Omron CX-Programmer project NewProject (CX-Programmer 9.73)

# PLC system: CP1L M

## Global symbols (name address type ; comment)
ALL_TANKS_ARE_FULL 102.04 BOOL  ; Cac thung day
AUTO 0.03 BOOL  ; Tu dong
C0004 BOOL  ; 1
D0 CHANNEL  ; COMPARE
D2 CHANNEL  ; .
BLOWER 100.00 BOOL  ; Lam sach
CHECK_1 1.10 BOOL  ; Kiem tra 1
CHECK_2 1.11 BOOL  ; Kiem tra 2
CHECK_3 2.00 BOOL  ; Kiem tra 3
CONVETOR_W2 101.02 BOOL  ; Chuyen doi 2
CONVEYOR_1 103.01 BOOL  ; Bang chuyen 1
CONVEYOR_10 103.09 BOOL  ; Bang chuyen 10
CONVEYOR_11 103.10 BOOL  ; Bang chuyen 11
CONVEYOR_2 103.02 BOOL  ; Bang chuyen 2
CONVEYOR_3 103.03 BOOL  ; Bang chuyen 3
CONVEYOR_5 103.04 BOOL  ; Bang chuyen 5
CONVEYOR_6 103.05 BOOL  ; Bang chuyen 6
CONVEYOR_7 103.06 BOOL  ; Bang chuyen 7
CONVEYOR_9 103.08 BOOL  ; Bang chuyen 9
CONVEYOR_W1 101.01 BOOL  ; Chuyen doi 1
CONVEYOR_W3 101.03 BOOL  ; Chuyen doi 3
DEFAULT_TANK_VOLUME 2.02 BOOL  ; Muc be mac dinh
DROP_1 101.04 BOOL  ; Tha 1
DROP_2 101.05 BOOL  ; Tha 2
DROP_3 101.06 BOOL  ; Tha 3
EJECT_BLOWER 100.01 BOOL  ; Ngung lam sach
EJECT_PRINT 100.04 BOOL  ; Ngung in
ERROR_LIGHT 101.00 BOOL  ; Den bao dong
KEEP_SENSOR_C1 102.03 BOOL  ; Giu cam bien 1
KEEP_SENSOR_C2 102.02 BOOL  ; Giu cam bien 2
KEEP_SENSOR_C3 102.01 BOOL  ; Giu cam bien 3
MANUAL 0.02 BOOL  ; In don chiec
METAL 2.06 BOOL  ; Kim loai
PAPER 2.07 BOOL  ; Giay
PLASTIC 2.08 BOOL  ; Nhua
POWER 103.00 BOOL  ; Nguon
PRINT_LIGHT 100.02 BOOL  ; In sang
PRINT_MACHINE 100.03 BOOL  ; In may
QUALITIFY_SENSOR 1.09 BOOL  ; Cam bien chat luong
REJECT 101.07 BOOL  ; Loai bo
REJECTED_PRODUCT 2.01 BOOL  ; San pham loi
REJECT_CONVEYOR 103.07 BOOL  ; Bang chuyen san pham loi
RESET_ALL 102.08 BOOL  ; Doi het cac thung
RESET_PACK_1 102.05 BOOL  ; Doi thung 1
RESET_PACK_2 102.06 BOOL  ; Doi thung 2
RESET_PACK_3 102.07 BOOL  ; Doi thung 3
ROBOT_CLA 102.00 BOOL  ; Canh tay robot
SENSOR_1 1.00 BOOL  ; Cam bien 1
SENSOR_2 1.01 BOOL  ; Cam bien 2
SENSOR_3 1.02 BOOL  ; Cam bien 3
SENSOR_4 1.03 BOOL  ; Cam bien 4
SENSOR_5 1.04 BOOL  ; Cam bien 5
SENSOR_6 1.05 BOOL  ; Cam bien 6
SENSOR_CLASSTIFY_1 1.08 BOOL  ; Cam bien phan loai 1
SENSOR_CLASSTIFY_2 1.07 BOOL  ; Cam bien phan loai 2
SENSOR_CLASSTIFY_3 1.06 BOOL  ; Cam bien phan loai 3
SENSOR_PACK_1 2.03 BOOL  ; Cam bien hang 1
SENSOR_PACK_2 2.04 BOOL  ; Cam bien hang 2
SENSOR_PACK_3 2.05 BOOL  ; Cam bien hang 3
START 0.00 BOOL  ; Nut khoi dong
STOP 0.01 BOOL  ; Nut dung
WAY_1 100.05 BOOL  ; Duong 1
WAY_2 100.06 BOOL  ; Duong 2
WAY_3 100.07 BOOL  ; Duong 3

## Program NewProgram1 (cyclic task 0)
Local symbols
dD0 UINT

### Section Section1

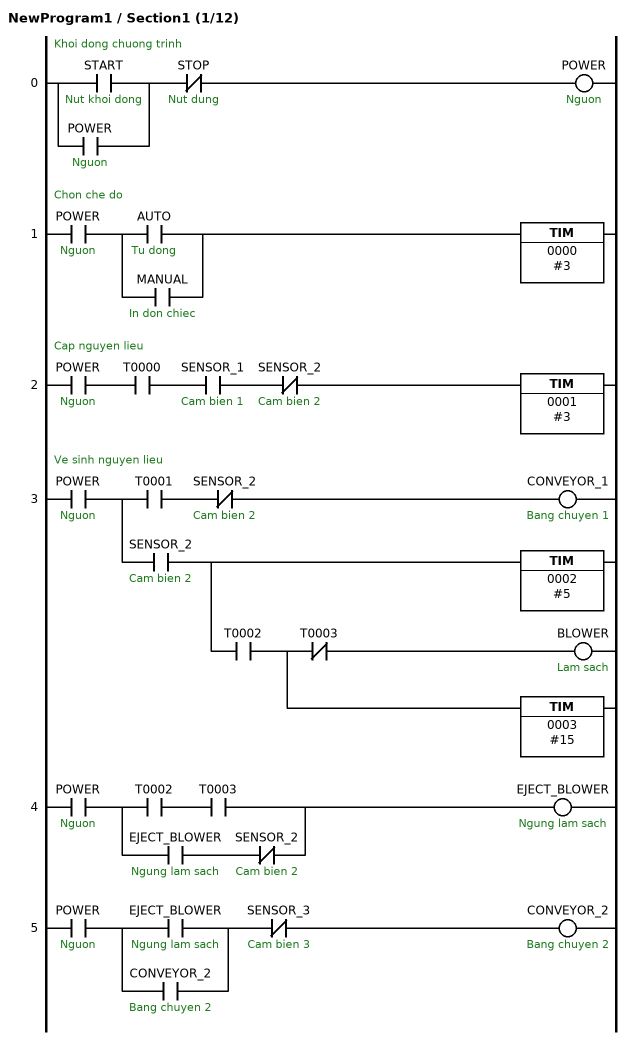
; rung 0: Khoi dong chuong trinh
LD START  ; Nut khoi dong
OR POWER  ; Nguon
ANDNOT STOP  ; Nut dung
OUT POWER  ; Nguon
; rung 1: Chon che do
LD POWER  ; Nguon
LD AUTO  ; Tu dong
OR MANUAL  ; In don chiec
ANDLD
TIM 0000 #3
; rung 2: Cap nguyen lieu
LD POWER  ; Nguon
AND T0000
AND SENSOR_1  ; Cam bien 1
ANDNOT SENSOR_2  ; Cam bien 2
TIM 0001 #3
; rung 3: Ve sinh nguyen lieu
LD POWER  ; Nguon
OUT TR0
AND T0001
ANDNOT SENSOR_2  ; Cam bien 2
OUT CONVEYOR_1  ; Bang chuyen 1
LD TR0
AND SENSOR_2  ; Cam bien 2
TIM 0002 #5
AND T0002
OUT TR0
ANDNOT T0003
OUT BLOWER  ; Lam sach
LD TR0
TIM 0003 #15
; rung 4
LD POWER  ; Nguon
LD T0002
AND T0003
LD EJECT_BLOWER  ; Ngung lam sach
ANDNOT SENSOR_2  ; Cam bien 2
ORLD
ANDLD
OUT EJECT_BLOWER  ; Ngung lam sach
; rung 5
LD POWER  ; Nguon
LD EJECT_BLOWER  ; Ngung lam sach
OR CONVEYOR_2  ; Bang chuyen 2
ANDLD
ANDNOT SENSOR_3  ; Cam bien 3
OUT CONVEYOR_2  ; Bang chuyen 2

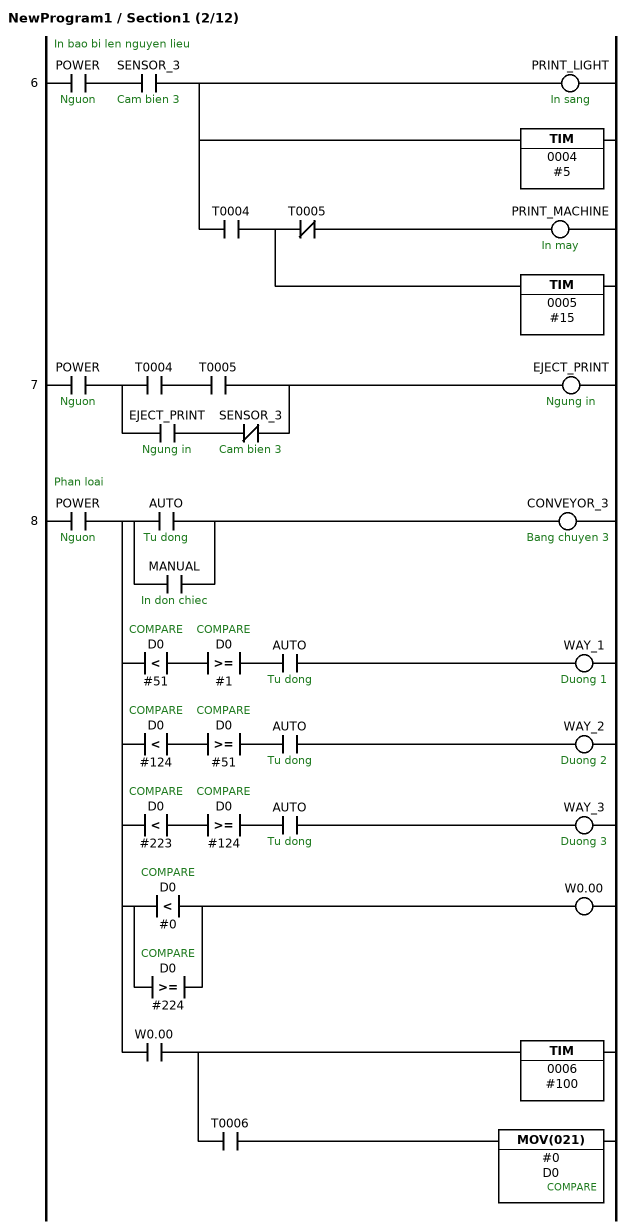
; rung 6: In bao bi len nguyen lieu
LD POWER  ; Nguon
AND SENSOR_3  ; Cam bien 3
OUT PRINT_LIGHT  ; In sang
TIM 0004 #5
AND T0004
OUT TR0
ANDNOT T0005
OUT PRINT_MACHINE  ; In may
LD TR0
TIM 0005 #15
; rung 7
LD POWER  ; Nguon
LD T0004
AND T0005
LD EJECT_PRINT  ; Ngung in
ANDNOT SENSOR_3  ; Cam bien 3
ORLD
ANDLD
OUT EJECT_PRINT  ; Ngung in
; rung 8: Phan loai
LD POWER  ; Nguon
OUT TR0
LD AUTO  ; Tu dong
OR MANUAL  ; In don chiec
ANDLD
OUT CONVEYOR_3  ; Bang chuyen 3
LD TR0
AND<(310) D0 #51  ; COMPARE
AND>=(325) D0 #1  ; COMPARE
AND AUTO  ; Tu dong
OUT WAY_1  ; Duong 1
LD TR0
AND<(310) D0 #124  ; COMPARE
AND>=(325) D0 #51  ; COMPARE
AND AUTO  ; Tu dong
OUT WAY_2  ; Duong 2
LD TR0
AND<(310) D0 #223  ; COMPARE
AND>=(325) D0 #124  ; COMPARE
AND AUTO  ; Tu dong
OUT WAY_3  ; Duong 3
LD TR0
LD<(310) D0 #0  ; COMPARE
OR>=(325) D0 #224  ; COMPARE
ANDLD
OUT W0.00
LD TR0
AND W0.00
TIM 0006 #100
AND T0006
MOV(021) #0 D0  ; COMPARE

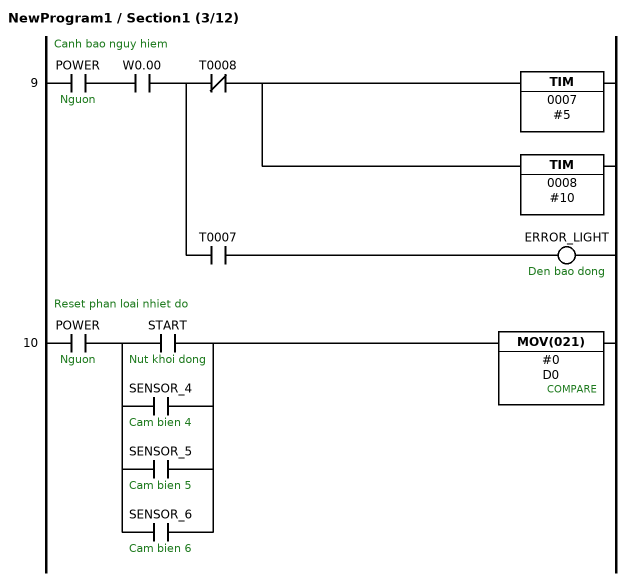
; rung 9: Canh bao nguy hiem
LD POWER  ; Nguon
AND W0.00
OUT TR0
ANDNOT T0008
TIM 0007 #5
TIM 0008 #10
LD TR0
AND T0007
OUT ERROR_LIGHT  ; Den bao dong
; rung 10: Reset phan loai nhiet do
LD POWER  ; Nguon
LD START  ; Nut khoi dong
OR SENSOR_4  ; Cam bien 4
OR SENSOR_5  ; Cam bien 5
OR SENSOR_6  ; Cam bien 6
ANDLD
MOV(021) #0 D0  ; COMPARE

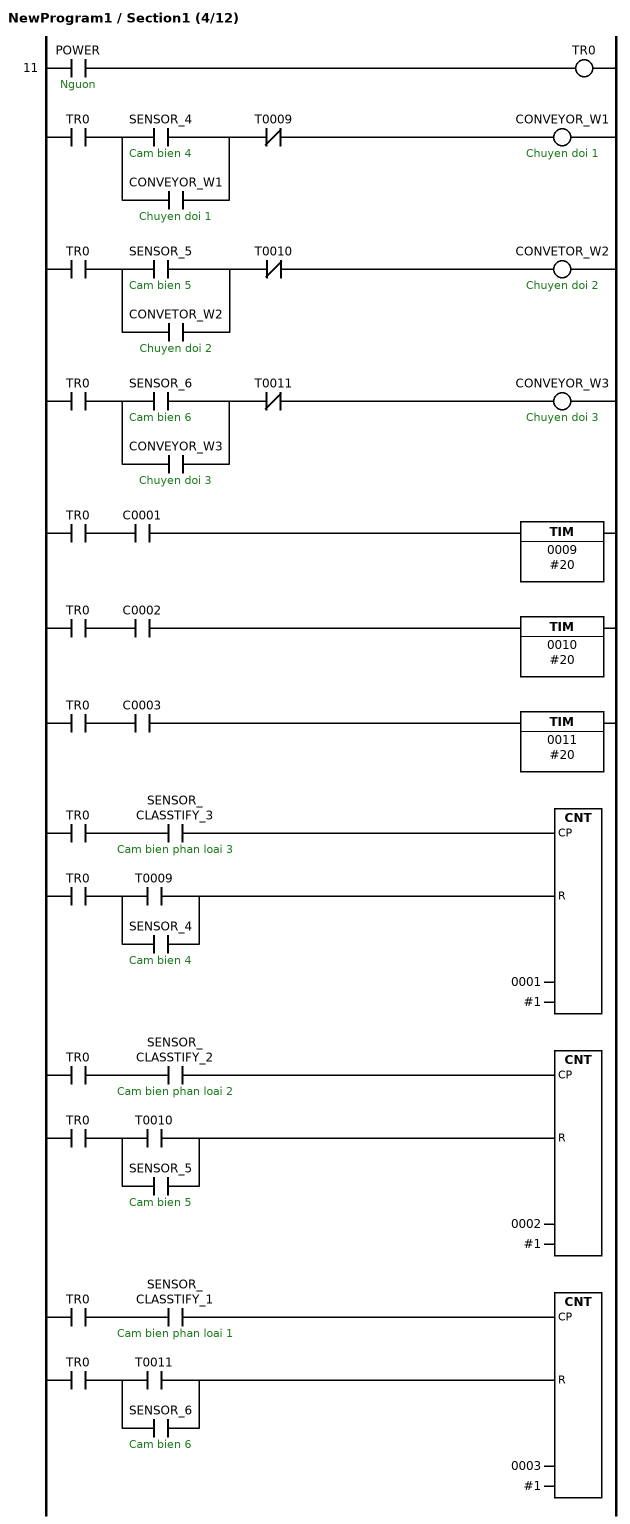
; rung 11
LD POWER  ; Nguon
OUT TR0
LD SENSOR_4  ; Cam bien 4
OR CONVEYOR_W1  ; Chuyen doi 1
ANDLD
ANDNOT T0009
OUT CONVEYOR_W1  ; Chuyen doi 1
LD TR0
LD SENSOR_5  ; Cam bien 5
OR CONVETOR_W2  ; Chuyen doi 2
ANDLD
ANDNOT T0010
OUT CONVETOR_W2  ; Chuyen doi 2
LD TR0
LD SENSOR_6  ; Cam bien 6
OR CONVEYOR_W3  ; Chuyen doi 3
ANDLD
ANDNOT T0011
OUT CONVEYOR_W3  ; Chuyen doi 3
LD TR0
AND C0001
TIM 0009 #20
LD TR0
AND C0002
TIM 0010 #20
LD TR0
AND C0003
TIM 0011 #20
LD TR0
AND SENSOR_CLASSTIFY_3  ; Cam bien phan loai 3
LD TR0
LD T0009
OR SENSOR_4  ; Cam bien 4
ANDLD
CNT 0001 #1
LD TR0
AND SENSOR_CLASSTIFY_2  ; Cam bien phan loai 2
LD TR0
LD T0010
OR SENSOR_5  ; Cam bien 5
ANDLD
CNT 0002 #1
LD TR0
AND SENSOR_CLASSTIFY_1  ; Cam bien phan loai 1
LD TR0
LD T0011
OR SENSOR_6  ; Cam bien 6
ANDLD
CNT 0003 #1

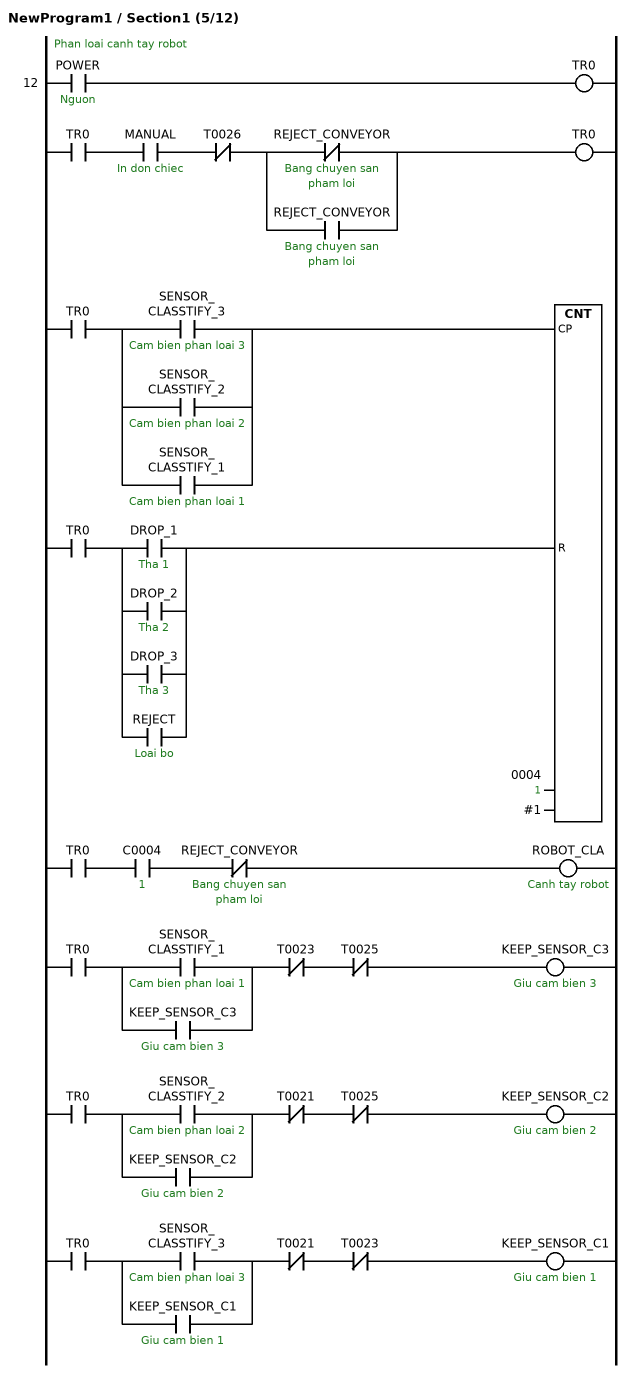
; rung 12: Phan loai canh tay robot
LD POWER  ; Nguon
OUT TR0
LD SENSOR_CLASSTIFY_3  ; Cam bien phan loai 3
OR SENSOR_CLASSTIFY_2  ; Cam bien phan loai 2
OR SENSOR_CLASSTIFY_1  ; Cam bien phan loai 1
ANDLD
LD TR0
LD DROP_1  ; Tha 1
OR DROP_2  ; Tha 2
OR DROP_3  ; Tha 3
OR REJECT  ; Loai bo
ANDLD
CNT 0004 #1  ; 1
LD TR0
AND C0004  ; 1
ANDNOT REJECT_CONVEYOR  ; Bang chuyen san pham loi
OUT ROBOT_CLA  ; Canh tay robot
LD TR0
AND MANUAL  ; In don chiec
ANDNOT T0026
LDNOT REJECT_CONVEYOR  ; Bang chuyen san pham loi
OR REJECT_CONVEYOR  ; Bang chuyen san pham loi
ANDLD
OUT TR0
LD SENSOR_CLASSTIFY_1  ; Cam bien phan loai 1
OR KEEP_SENSOR_C3  ; Giu cam bien 3
ANDLD
ANDNOT T0023
ANDNOT T0025
OUT KEEP_SENSOR_C3  ; Giu cam bien 3
LD TR0
LD SENSOR_CLASSTIFY_2  ; Cam bien phan loai 2
OR KEEP_SENSOR_C2  ; Giu cam bien 2
ANDLD
ANDNOT T0021
ANDNOT T0025
OUT KEEP_SENSOR_C2  ; Giu cam bien 2
LD TR0
LD SENSOR_CLASSTIFY_3  ; Cam bien phan loai 3
OR KEEP_SENSOR_C1  ; Giu cam bien 1
ANDLD
ANDNOT T0021
ANDNOT T0023
OUT KEEP_SENSOR_C1  ; Giu cam bien 1

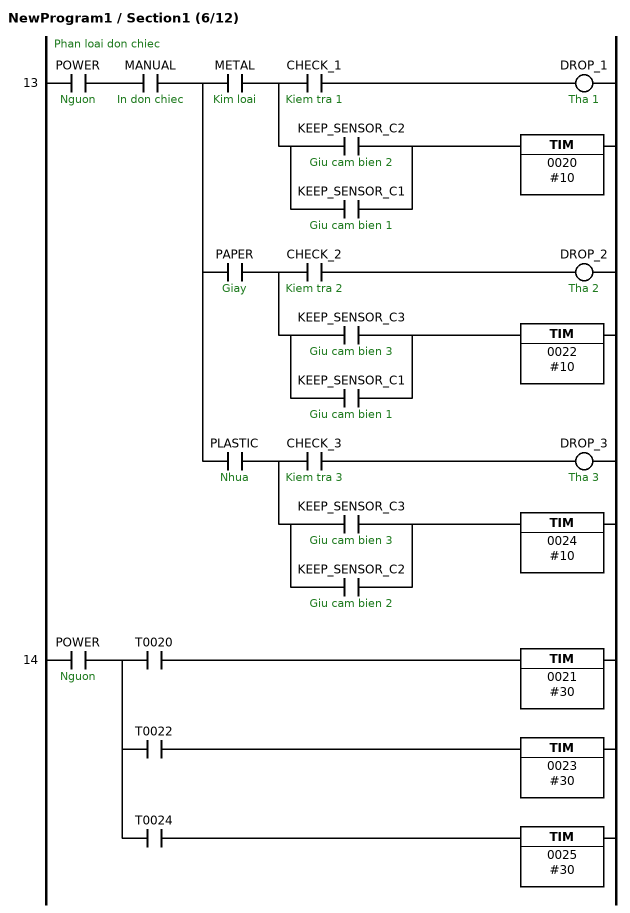
; rung 13: Phan loai don chiec
LD POWER  ; Nguon
AND MANUAL  ; In don chiec
OUT TR0
AND METAL  ; Kim loai
OUT TR1
AND CHECK_1  ; Kiem tra 1
OUT DROP_1  ; Tha 1
LD TR1
LD KEEP_SENSOR_C2  ; Giu cam bien 2
OR KEEP_SENSOR_C1  ; Giu cam bien 1
ANDLD
TIM 0020 #10
LD TR0
AND PAPER  ; Giay
OUT TR1
AND CHECK_2  ; Kiem tra 2
OUT DROP_2  ; Tha 2
LD TR1
LD KEEP_SENSOR_C3  ; Giu cam bien 3
OR KEEP_SENSOR_C1  ; Giu cam bien 1
ANDLD
TIM 0022 #10
LD TR0
AND PLASTIC  ; Nhua
OUT TR0
AND CHECK_3  ; Kiem tra 3
OUT DROP_3  ; Tha 3
LD TR0
LD KEEP_SENSOR_C3  ; Giu cam bien 3
OR KEEP_SENSOR_C2  ; Giu cam bien 2
ANDLD
TIM 0024 #10
; rung 14
LD POWER  ; Nguon
OUT TR0
AND T0020
TIM 0021 #30
LD TR0
AND T0022
TIM 0023 #30
LD TR0
AND T0024
TIM 0025 #30

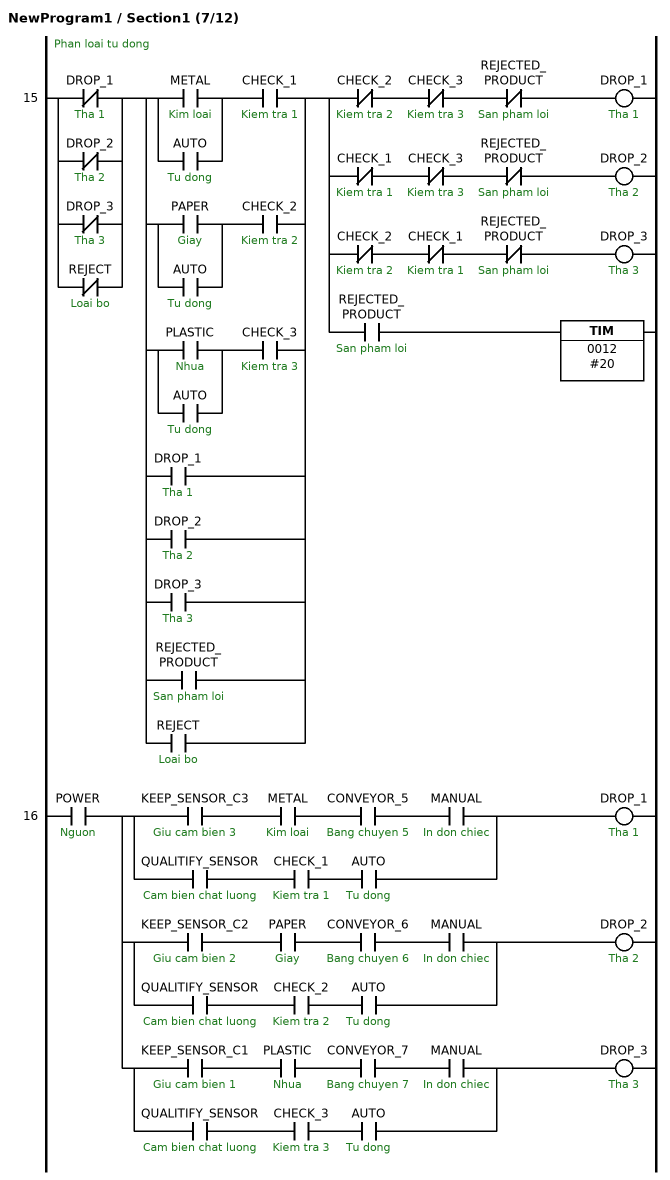
; rung 15: Phan loai tu dong
LDNOT DROP_1  ; Tha 1
ORNOT DROP_2  ; Tha 2
ORNOT DROP_3  ; Tha 3
ORNOT REJECT  ; Loai bo
LD METAL  ; Kim loai
OR AUTO  ; Tu dong
AND CHECK_1  ; Kiem tra 1
LD PAPER  ; Giay
OR AUTO  ; Tu dong
AND CHECK_2  ; Kiem tra 2
ORLD
LD PLASTIC  ; Nhua
OR AUTO  ; Tu dong
AND CHECK_3  ; Kiem tra 3
ORLD
OR DROP_1  ; Tha 1
OR DROP_2  ; Tha 2
OR DROP_3  ; Tha 3
OR REJECTED_PRODUCT  ; San pham loi
OR REJECT  ; Loai bo
ANDLD
OUT TR0
ANDNOT CHECK_2  ; Kiem tra 2
ANDNOT CHECK_3  ; Kiem tra 3
ANDNOT REJECTED_PRODUCT  ; San pham loi
OUT DROP_1  ; Tha 1
LD TR0
ANDNOT CHECK_1  ; Kiem tra 1
ANDNOT CHECK_3  ; Kiem tra 3
ANDNOT REJECTED_PRODUCT  ; San pham loi
OUT DROP_2  ; Tha 2
LD TR0
ANDNOT CHECK_2  ; Kiem tra 2
ANDNOT CHECK_1  ; Kiem tra 1
ANDNOT REJECTED_PRODUCT  ; San pham loi
OUT DROP_3  ; Tha 3
LD TR0
AND REJECTED_PRODUCT  ; San pham loi
TIM 0012 #20
; rung 16
LD POWER  ; Nguon
OUT TR0
LD KEEP_SENSOR_C3  ; Giu cam bien 3
AND METAL  ; Kim loai
AND CONVEYOR_5  ; Bang chuyen 5
AND MANUAL  ; In don chiec
LD QUALITIFY_SENSOR  ; Cam bien chat luong
AND CHECK_1  ; Kiem tra 1
AND AUTO  ; Tu dong
ORLD
ANDLD
OUT DROP_1  ; Tha 1
LD TR0
LD KEEP_SENSOR_C2  ; Giu cam bien 2
AND PAPER  ; Giay
AND CONVEYOR_6  ; Bang chuyen 6
AND MANUAL  ; In don chiec
LD QUALITIFY_SENSOR  ; Cam bien chat luong
AND CHECK_2  ; Kiem tra 2
AND AUTO  ; Tu dong
ORLD
ANDLD
OUT DROP_2  ; Tha 2
LD TR0
LD KEEP_SENSOR_C1  ; Giu cam bien 1
AND PLASTIC  ; Nhua
AND CONVEYOR_7  ; Bang chuyen 7
AND MANUAL  ; In don chiec
LD QUALITIFY_SENSOR  ; Cam bien chat luong
AND CHECK_3  ; Kiem tra 3
AND AUTO  ; Tu dong
ORLD
ANDLD
OUT DROP_3  ; Tha 3

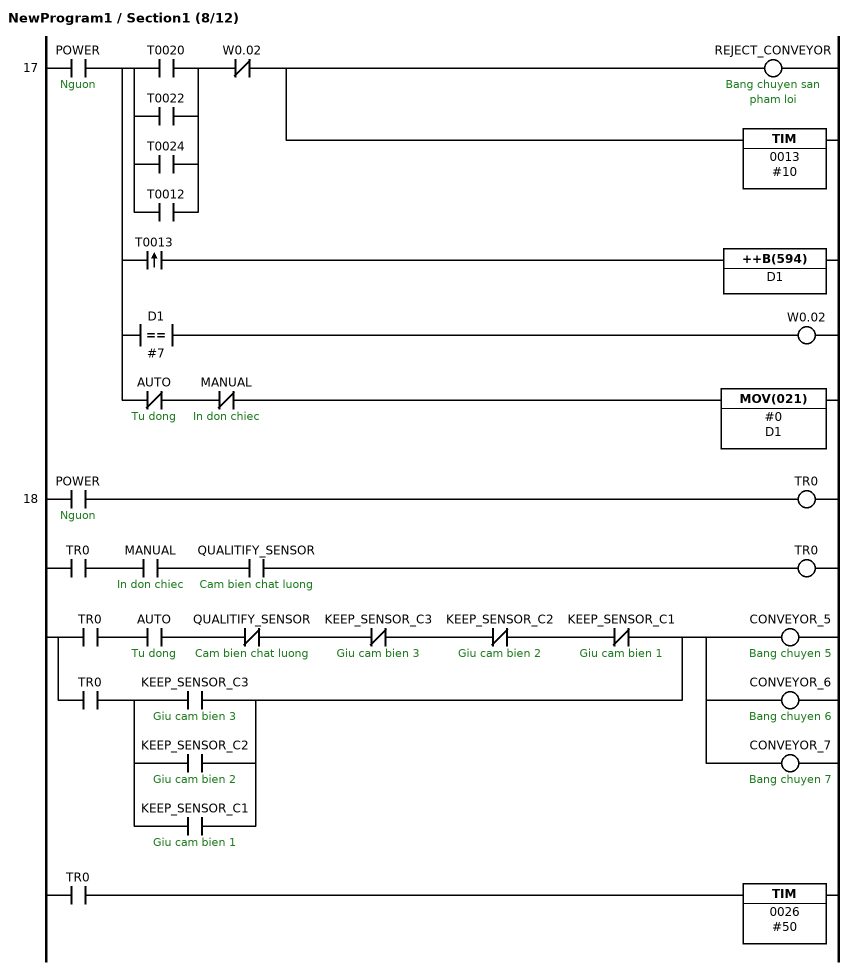
; rung 17
LD POWER  ; Nguon
OUT TR0
LD T0020
OR T0022
OR T0024
OR T0012
ANDLD
ANDNOT W0.02
OUT REJECT_CONVEYOR  ; Bang chuyen san pham loi
TIM 0013 #10
LD TR0
@AND T0013
++B(594) D1
LD TR0
AND=(300) D1 #7
OUT W0.02
LD TR0
ANDNOT AUTO  ; Tu dong
ANDNOT MANUAL  ; In don chiec
MOV(021) #0 D1
; rung 18
LD POWER  ; Nguon
OUT TR0
AND AUTO  ; Tu dong
ANDNOT QUALITIFY_SENSOR  ; Cam bien chat luong
ANDNOT KEEP_SENSOR_C3  ; Giu cam bien 3
ANDNOT KEEP_SENSOR_C2  ; Giu cam bien 2
ANDNOT KEEP_SENSOR_C1  ; Giu cam bien 1
LD TR0
AND MANUAL  ; In don chiec
AND QUALITIFY_SENSOR  ; Cam bien chat luong
OUT TR0
LD KEEP_SENSOR_C3  ; Giu cam bien 3
OR KEEP_SENSOR_C2  ; Giu cam bien 2
OR KEEP_SENSOR_C1  ; Giu cam bien 1
ANDLD
ORLD
OUT CONVEYOR_5  ; Bang chuyen 5
OUT CONVEYOR_6  ; Bang chuyen 6
OUT CONVEYOR_7  ; Bang chuyen 7
LD TR0
TIM 0026 #50

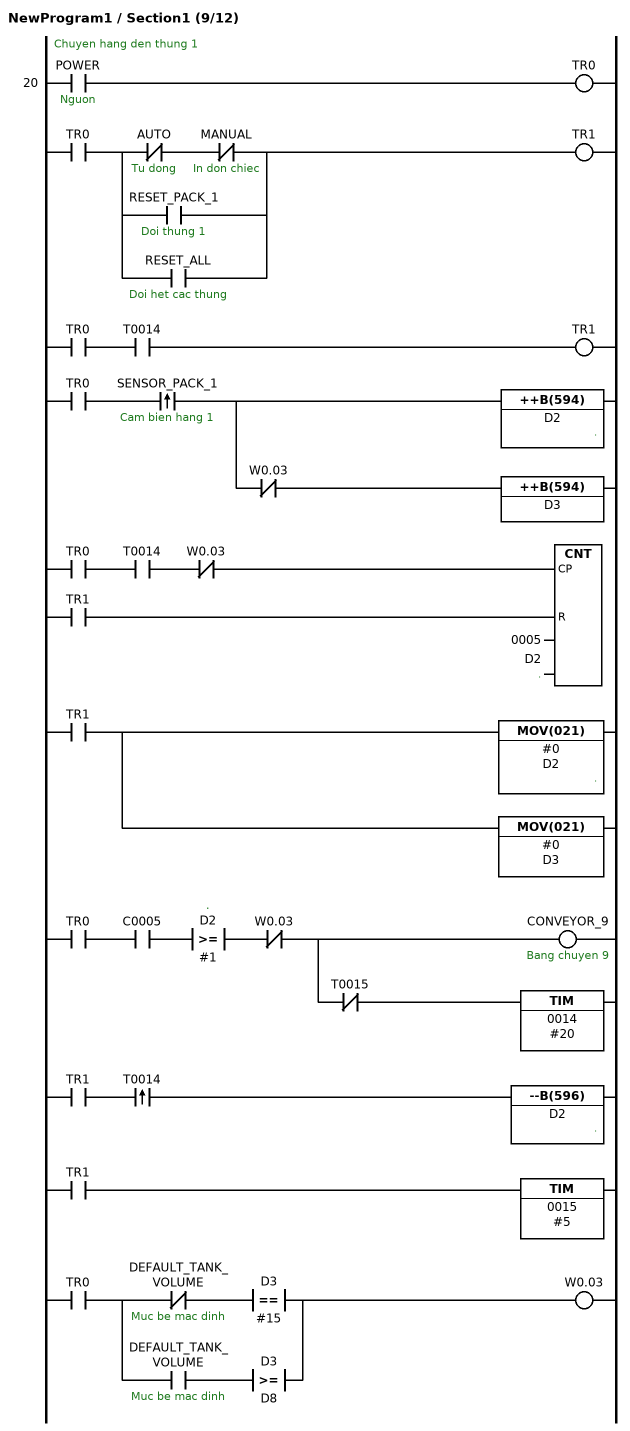
; rung 20: Chuyen hang den thung 1
LD POWER  ; Nguon
OUT TR0
@AND SENSOR_PACK_1  ; Cam bien hang 1
++B(594) D2  ; .
ANDNOT W0.03
++B(594) D3
LD TR0
AND T0014
ANDNOT W0.03
LD TR0
LDNOT AUTO  ; Tu dong
ANDNOT MANUAL  ; In don chiec
OR RESET_PACK_1  ; Doi thung 1
OR RESET_ALL  ; Doi het cac thung
ANDLD
OUT TR1
CNT 0005 D2  ; .
LD TR1
MOV(021) #0 D2  ; .
MOV(021) #0 D3
LD TR0
AND C0005
AND>=(325) D2 #1  ; .
ANDNOT W0.03
OUT CONVEYOR_9  ; Bang chuyen 9
ANDNOT T0015
TIM 0014 #20
LD TR0
AND T0014
OUT TR1
@AND T0014
--B(596) D2  ; .
LD TR1
TIM 0015 #5
LD TR0
LDNOT DEFAULT_TANK_VOLUME  ; Muc be mac dinh
AND=(300) D3 #15
LD DEFAULT_TANK_VOLUME  ; Muc be mac dinh
AND>=(325) D3 D8
ORLD
ANDLD
OUT W0.03

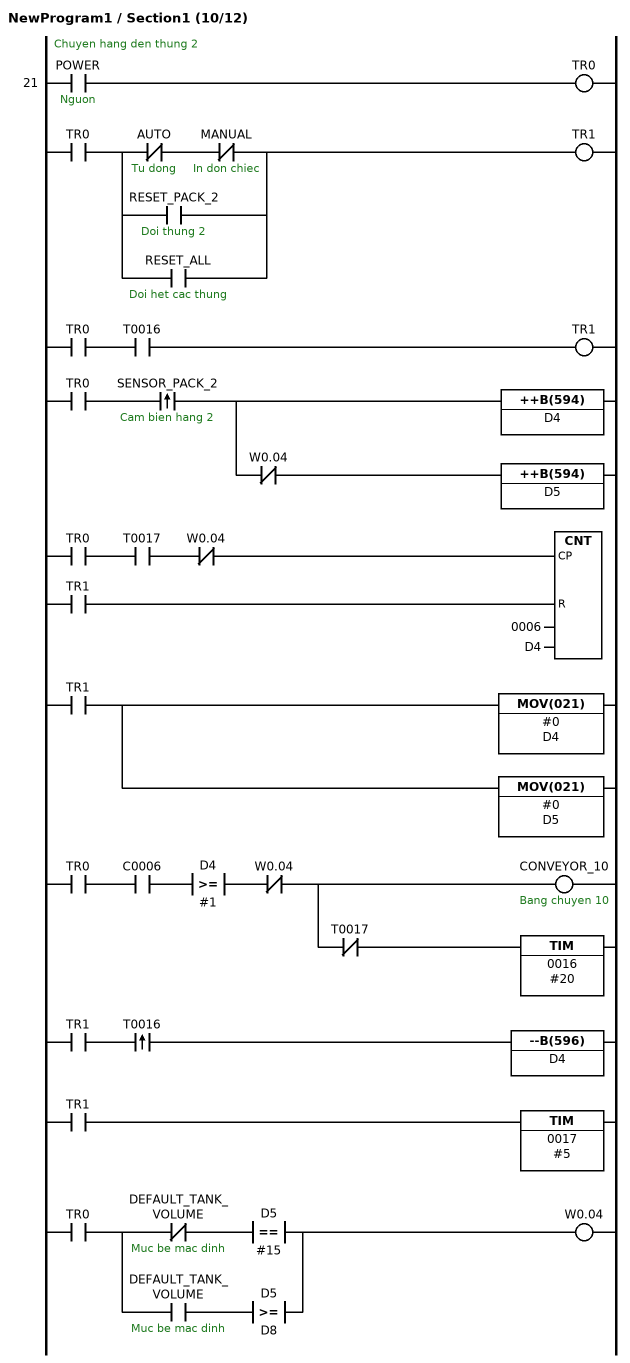
; rung 21: Chuyen hang den thung 2
LD POWER  ; Nguon
OUT TR0
@AND SENSOR_PACK_2  ; Cam bien hang 2
++B(594) D4
ANDNOT W0.04
++B(594) D5
LD TR0
AND T0017
ANDNOT W0.04
LD TR0
LDNOT AUTO  ; Tu dong
ANDNOT MANUAL  ; In don chiec
OR RESET_PACK_2  ; Doi thung 2
OR RESET_ALL  ; Doi het cac thung
ANDLD
OUT TR1
CNT 0006 D4
LD TR1
MOV(021) #0 D4
MOV(021) #0 D5
LD TR0
AND C0006
AND>=(325) D4 #1
ANDNOT W0.04
OUT CONVEYOR_10  ; Bang chuyen 10
ANDNOT T0017
TIM 0016 #20
LD TR0
AND T0016
OUT TR1
@AND T0016
--B(596) D4
LD TR1
TIM 0017 #5
LD TR0
LDNOT DEFAULT_TANK_VOLUME  ; Muc be mac dinh
AND=(300) D5 #15
LD DEFAULT_TANK_VOLUME  ; Muc be mac dinh
AND>=(325) D5 D8
ORLD
ANDLD
OUT W0.04

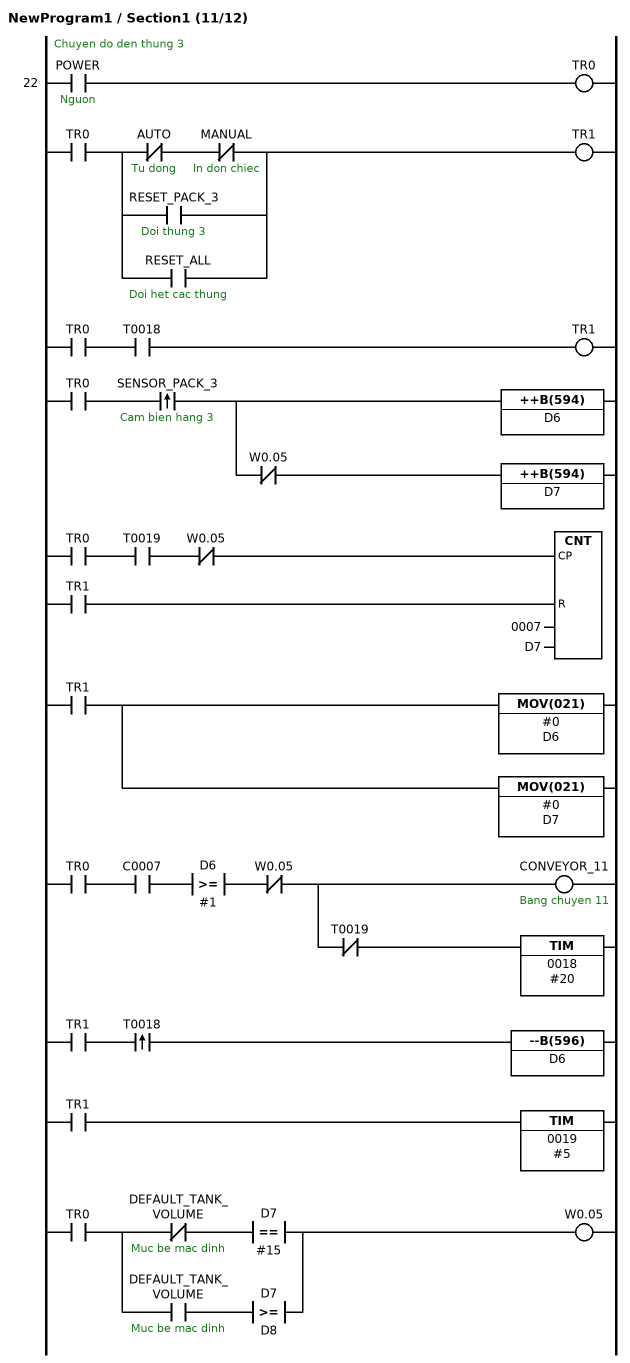
; rung 22: Chuyen do den thung 3
LD POWER  ; Nguon
OUT TR0
@AND SENSOR_PACK_3  ; Cam bien hang 3
++B(594) D6
ANDNOT W0.05
++B(594) D7
LD TR0
AND T0019
ANDNOT W0.05
LD TR0
LDNOT AUTO  ; Tu dong
ANDNOT MANUAL  ; In don chiec
OR RESET_PACK_3  ; Doi thung 3
OR RESET_ALL  ; Doi het cac thung
ANDLD
OUT TR1
CNT 0007 D7
LD TR1
MOV(021) #0 D6
MOV(021) #0 D7
LD TR0
AND C0007
AND>=(325) D6 #1
ANDNOT W0.05
OUT CONVEYOR_11  ; Bang chuyen 11
ANDNOT T0019
TIM 0018 #20
LD TR0
AND T0018
OUT TR1
@AND T0018
--B(596) D6
LD TR1
TIM 0019 #5
LD TR0
LDNOT DEFAULT_TANK_VOLUME  ; Muc be mac dinh
AND=(300) D7 #15
LD DEFAULT_TANK_VOLUME  ; Muc be mac dinh
AND>=(325) D7 D8
ORLD
ANDLD
OUT W0.05

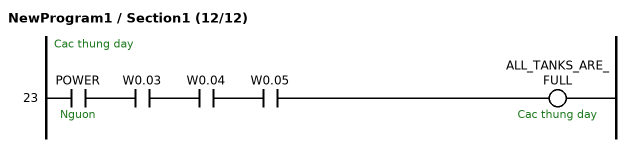
; rung 23: Cac thung day
LD POWER  ; Nguon
AND W0.03
AND W0.04
AND W0.05
OUT ALL_TANKS_ARE_FULL  ; Cac thung day

### Section END
; rung 0
END(001)